// TwinCAT 3 PLC project Database_Connection
// ProgramVersion: 3.1.4026.14
// libraries:
//   Tc2_Standard, * (Beckhoff Automation GmbH)
//   Tc2_System, * (Beckhoff Automation GmbH)
//   Tc3_Database, * (Beckhoff Automation GmbH)
//   Tc3_EventLogger, * (Beckhoff Automation GmbH)
// project tree:
//   DUTs/ DUT_SQL.TcDUT
//   / PlcTask.TcTTO
//   POUs/ MAIN.TcPOU (not stored), FC_SQL_InsertCommands.TcPOU (not stored)
// real-time tasks:
//   TASK PlcTask: cycle T#10ms, priority 20, ADS port 350

CONFIGURATION Database_Connection
    RESOURCE PLC ON TwinCAT3
        TASK PlcTask(INTERVAL := T#10ms, PRIORITY := 20);
        PROGRAM MAIN WITH PlcTask : MAIN;
    END_RESOURCE
END_CONFIGURATION

// ---- DUTs/DUT_SQL.TcDUT
TYPE DUT_SQL :
STRUCT
    SensorValue : INT;
    SampleNr : INT;
    Timestamp : STRING(50);
END_STRUCT
END_TYPE
